FUNCTION_BLOCK FB86
TITLE = 'pilot'
AUTHOR : CB

VAR
	pilot_F1 : FB74;
	pilot_F2 : FB80;
	pilot_F3 : FB84;
END_VAR


BEGIN


NETWORK
TITLE =
//
//	pilot/pilot_F1
CALL #pilot_F1;



NETWORK
TITLE =
//
//	pilot/pilot_F2
CALL #pilot_F2;



NETWORK
TITLE =
//
//	pilot/pilot_F3
CALL #pilot_F3;




END_FUNCTION_BLOCK
